INTERFACE I_Mover

METHOD Mover : REAL
VAR_INPUT
	Velocidad_Deseada : REAL;
END_VAR
END_METHOD

END_INTERFACE

(* stored: Version 1.1.0.1, ProductVersion 3.1.4024.12
   Itf I_Mover: Id {110b19c7-99f3-4443-957d-3705f79b94ec}
   Method Mover: Id {e24c3df2-6b95-4e7f-bd0f-786760ff5bbb} *)
